FUNCTION_BLOCK Pneumatic_1Coil_Management
// Function block untuk mengolah faceplate dan watchdog pneumatic valve 1 coil
//	UDT dependencies:
	(*  
	1. stPneumatic v1.0 	*)

//	Changelog:
	(* 
	v1.0 [27.12.2021] Start development function block - Fabrilian Asali	*)	

VAR_INPUT
	bEnable						: BOOL;		
	bTriggerPneumatic			: BOOL;
	bTestMode					: BOOL;
	bResetError					: BOOL;
	bBypassSensorRetract		: BOOL;
	bBypassSensorAdvanced		: BOOL;
	bBypassPreCheckSensor		: BOOL;
	xIn_SensorRetract			: BOOL;
	xIn_SensorAdvanced			: BOOL;
	TimerBypassSensorRetract	: TIME := T#5S;
	TimerBypassSensorAdvanced	: TIME := T#5S;
	TimerWatchdogRetract		: TIME := T#5S;
	TimerWatchdogAdvanced		: TIME := T#5S;
	TimerWatchdogPreRetract		: TIME := T#5S;
	TimerWatchdogPreAdvanced	: TIME := T#5S;
END_VAR

VAR_OUTPUT
	bError						: BOOL;
	ErrorID						: INT;
	ErrorMsg					: STRING;
END_VAR

VAR_IN_OUT
	Pneumatic					: stPneumatic1;
END_VAR

VAR
	SeqIndex					: INT;
	WatchdogTimer				: TON;
	bTrig_Output				: BOOL;
	PneuAdv						: R_TRIG;
	TimerBypass					: TON;
END_VAR
VAR // added by the converter: edge detectors and wires of the graphical bodies
    _rt1 : R_TRIG;
END_VAR

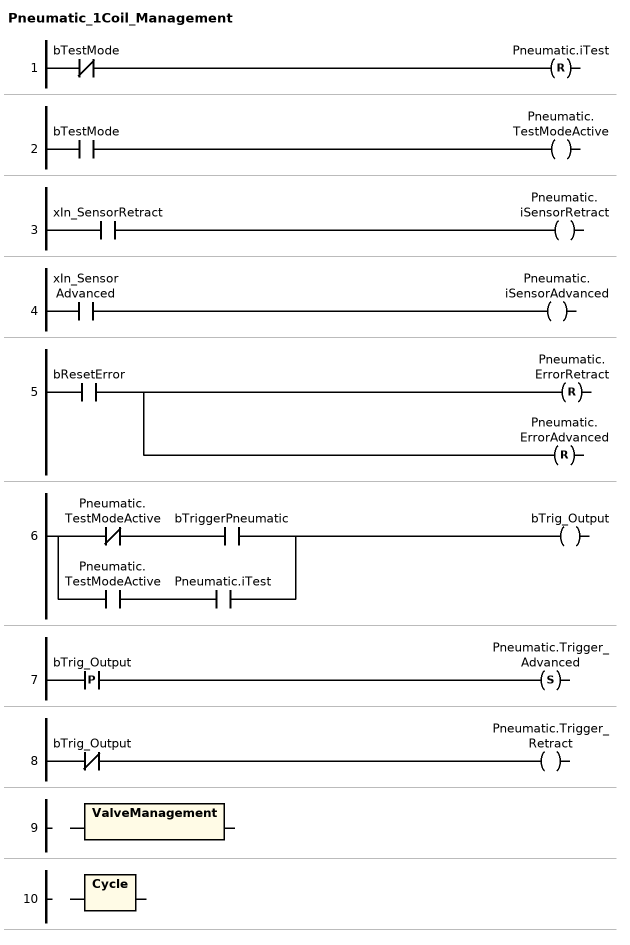
// NETWORK 1
Pneumatic.iTest R= NOT bTestMode;

// NETWORK 2
Pneumatic.TestModeActive := bTestMode;

// NETWORK 3
Pneumatic.iSensorRetract := xIn_SensorRetract;

// NETWORK 4
Pneumatic.iSensorAdvanced := xIn_SensorAdvanced;

// NETWORK 5
Pneumatic.ErrorRetract R= bResetError;
Pneumatic.ErrorAdvanced R= bResetError;

// NETWORK 6
bTrig_Output := NOT Pneumatic.TestModeActive AND bTriggerPneumatic OR Pneumatic.TestModeActive AND Pneumatic.iTest;

// NETWORK 7
_rt1(CLK := bTrig_Output);
Pneumatic.Trigger_Advanced S= _rt1.Q;

// NETWORK 8
Pneumatic.Trigger_Retract := NOT bTrig_Output;

// NETWORK 9
ValveManagement();

// NETWORK 10
Cycle();

ACTION Cycle:
PneuAdv (Clk := Pneumatic.oPneumatic);
IF PneuAdv.Q THEN
	Pneumatic.CyclePneu	:= Pneumatic.CyclePneu + 1;
END_IF
END_ACTION

ACTION ValveManagement:
IF bResetError THEN
	SeqIndex	:= 0;
	ErrorID		:= 0;
	ErrorMsg	:= '';
	bError		:= FALSE;
END_IF;

IF (bEnable OR Pneumatic.TestModeActive ) AND NOT bError THEN
	CASE SeqIndex OF
		0:
			WatchdogTimer(In:= FALSE);
			IF Pneumatic.Trigger_Retract AND NOT Pneumatic.FBDone_Retract THEN
				Pneumatic.FBDone_Retract:=FALSE;
				Pneumatic.FBDone_Advanced:=FALSE;
				SeqIndex	:= 100;
			ELSIF Pneumatic.Trigger_Advanced THEN
				Pneumatic.FBDone_Retract:=FALSE;
				Pneumatic.FBDone_Advanced:=FALSE;
				SeqIndex	:= 200;
			END_IF;
		
		100:
			Pneumatic.Trigger_Retract	:= FALSE;
			IF NOT bBypassPreCheckSensor THEN
				WatchdogTimer(In:= TRUE, PT:= TimerWatchdogPreRetract);
				IF Pneumatic.iSensorAdvanced THEN
					WatchdogTimer(In:= FALSE);
					SeqIndex	:= 110;
				ELSIF WatchdogTimer.Q THEN
					WatchdogTimer(In:= FALSE);
					Pneumatic.ErrorRetract := TRUE;
					ErrorID					:= 10;
					ErrorMsg				:= 'Error PreCheck Retract';
					SeqIndex	:= 999;
				END_IF;
			ELSE
				SeqIndex	:= 110;
			END_IF;
	
		110:
			Pneumatic.oPneumatic := FALSE;
			IF NOT bBypassSensorRetract THEN
				WatchdogTimer(In:= TRUE, PT:= TimerWatchdogRetract);
				IF Pneumatic.iSensorRetract THEN
					Pneumatic.FBDone_Retract:=TRUE;
					WatchdogTimer(In:= FALSE);
					SeqIndex	:= 0;
				ELSIF WatchdogTimer.Q THEN
					WatchdogTimer(In:= FALSE);
					Pneumatic.ErrorRetract := TRUE;
					ErrorID					:= 11;
					ErrorMsg				:= 'Error Watchdog Retract';
				END_IF;
			ELSE
				TimerBypass(In:= TRUE, PT:= TimerBypassSensorRetract);
				IF TimerBypass.Q THEN
					Pneumatic.FBDone_Retract:=TRUE;
					TimerBypass(In:= FALSE);
					SeqIndex	:= 0;
				END_IF;
			END_IF;
			
		200:
			Pneumatic.Trigger_Advanced	:= FALSE;
			IF NOT bBypassPreCheckSensor THEN
				WatchdogTimer(In:= TRUE, PT:= TimerWatchdogPreAdvanced);
				IF Pneumatic.iSensorRetract THEN
					WatchdogTimer(In:= FALSE);
					SeqIndex	:= 210;
				ELSIF WatchdogTimer.Q THEN
					WatchdogTimer(In:= FALSE);
					Pneumatic.ErrorAdvanced := TRUE;
					ErrorID					:= 20;
					ErrorMsg				:= 'Error PreCheck Advanced';
					SeqIndex	:= 999;
				END_IF;
			ELSE
				SeqIndex	:= 210;
			END_IF;				
		
		210:
			Pneumatic.oPneumatic := TRUE;
			IF NOT bBypassSensorAdvanced THEN
				WatchdogTimer(In:= TRUE, PT:= TimerWatchdogAdvanced);
				IF Pneumatic.iSensorAdvanced THEN
					Pneumatic.FBDone_Advanced:=TRUE;
					WatchdogTimer(In:= FALSE);
					SeqIndex	:= 0;
				ELSIF WatchdogTimer.Q THEN
					WatchdogTimer(In:= FALSE);
					Pneumatic.ErrorAdvanced := TRUE;
					ErrorID					:= 21;
					ErrorMsg				:= 'Error Watchdog Advanced';
				END_IF;
			ELSE
				TimerBypass(In:= TRUE, PT:= TimerBypassSensorAdvanced);
				IF TimerBypass.Q THEN
					Pneumatic.FBDone_Advanced:=TRUE;
					TimerBypass(In:= FALSE);
					SeqIndex	:= 0;
				END_IF;
				
			END_IF	;				
	
		999:
			bError	:= TRUE;	
			
	END_CASE;
ELSE
	IF bError OR Pneumatic.TestModeActive THEN
		SeqIndex := 0;
	END_IF;
	WatchdogTimer(IN:= FALSE);
	Pneumatic.Trigger_Advanced	:= FALSE;
	Pneumatic.Trigger_Retract	:= FALSE;
	Pneumatic.FBDone_Retract	:= FALSE;
	Pneumatic.FBDone_Advanced	:= FALSE;
END_IF;
END_ACTION

END_FUNCTION_BLOCK

(* stored: Version 1.1.0.1, ProductVersion 3.1.4024.12
   POU Pneumatic_1Coil_Management: Id {ccb4f153-69e5-4b35-b246-b531fd5cf5e3}, SpecialFunc None
   Action Cycle: Id {3b80401e-da04-4389-a863-a469b7bff54b}
   Action ValveManagement: Id {841fccbe-1ad3-4ca7-a1f5-b8b3ff32283d} *)
